// TIA Portal project "Practica_7_p2" (V14)

(* hardware
DEVICE "S7-1200 station_1"  S7-1200 Station
   slot 0: "Rack_0"  S7-1200 Rack  Rack  V1.0
   slot 1: "PLC_1"  CPU 1214C DC/DC/DC  6ES7 214-1AG40-0XB0  V4.2
*)

// ===== PLC "PLC_1"  CPU 1214C DC/DC/DC =====

VAR_GLOBAL   // PLC tag table "Default tag table"
   "G" AT %M0.0 : Bool;
   "R" AT %M0.1 : Bool;
   "LUZ_ROJA" AT %Q0.0 : Bool;
   "LUZ_VERDE" AT %Q0.1 : Bool;
   "OFF" AT %M0.2 : Bool;
   "PM" AT %I0.0 : Bool;
   "PP" AT %I0.1 : Bool;
   "EN" AT %M0.4 : Bool;
END_VAR

DATA_BLOCK "DB_TIMERS_CONFIG"   // DB1
{ S7_Optimized_Access := 'TRUE' }
VERSION : 0.1
   VAR
      TR : Time := T#6s;
      TV : Time := T#5s;
   END_VAR
BEGIN
END_DATA_BLOCK

// folder: System blocks/Program resources

DATA_BLOCK "t_r2v"   // DB2
{ S7_Optimized_Access := 'TRUE' }
AUTHOR : Simatic
FAMILY : IEC
NAME : IEC_TMR
VERSION : 1.0
// stored: InstanceOfName IEC_TIMER
"IEC_TIMER"
BEGIN
END_DATA_BLOCK

DATA_BLOCK "t_v2r"   // DB3
{ S7_Optimized_Access := 'TRUE' }
AUTHOR : Simatic
FAMILY : IEC
NAME : IEC_TMR
VERSION : 1.0
// stored: InstanceOfName IEC_TIMER
"IEC_TIMER"
BEGIN
END_DATA_BLOCK

// folder: (top level)

FUNCTION "FC_SEMAFORO_V1" : Void   // FC1, LAD
{ S7_Optimized_Access := 'TRUE' }
VERSION : 0.1
   VAR_INPUT
      ENABLE : Bool;
      TV : Time;
      TR : Time;
   END_VAR
   VAR_OUTPUT
      LR : Bool;
      LV : Bool;
   END_VAR
   VAR_TEMP   // added for the SCL form of the ladder/FBD networks
      _w1 : Bool;
      _w2 : Bool;
   END_VAR
BEGIN

REGION Network 1
   // INICIALIZACIÓN DE ESTADOS
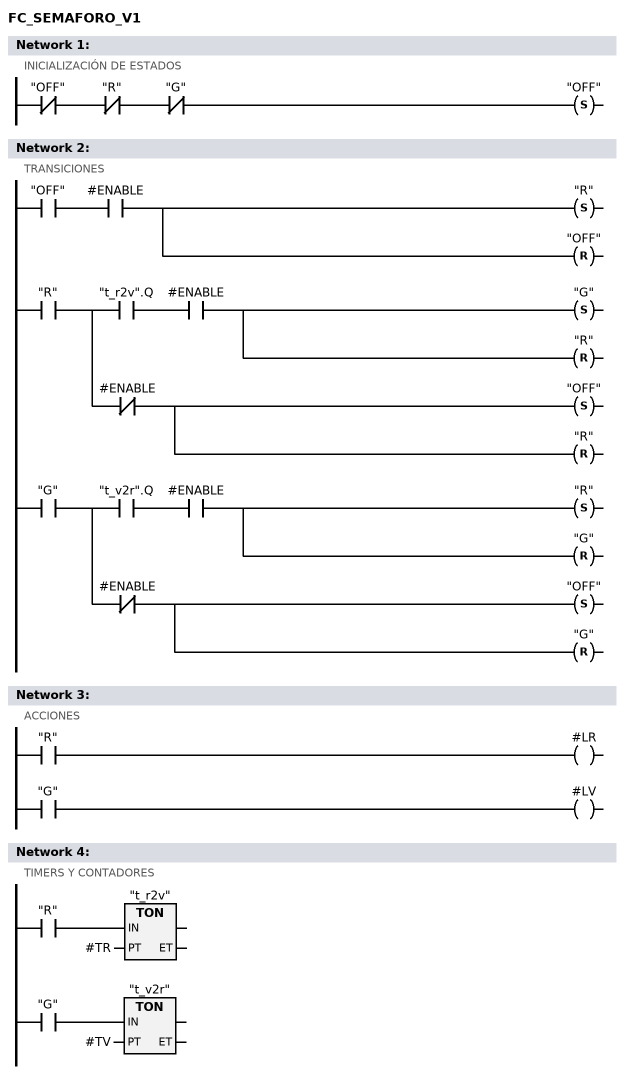
   RUNG wire#powerrail
      I_Contact( "OFF" )
      I_Contact( "R" )
      I_Contact( "G" )
      S_Coil( "OFF" )
   END_RUNG
   // the same network as SCL:
   IF NOT "OFF" AND NOT "R" AND NOT "G" THEN "OFF" := TRUE; END_IF;
END_REGION

REGION Network 2
   // TRANSICIONES
   RUNG wire#powerrail
      Contact( "OFF" )
      Contact( #ENABLE )
      wire#w1
      S_Coil( "R" )
   END_RUNG
   RUNG wire#w1
      R_Coil( "OFF" )
   END_RUNG
   RUNG wire#powerrail
      Contact( "R" )
      wire#w2
      Contact( "t_r2v".Q )
      Contact( #ENABLE )
      wire#w3
      S_Coil( "G" )
   END_RUNG
   RUNG wire#w3
      R_Coil( "R" )
   END_RUNG
   RUNG wire#w2
      I_Contact( #ENABLE )
      wire#w4
      S_Coil( "OFF" )
   END_RUNG
   RUNG wire#w4
      R_Coil( "R" )
   END_RUNG
   RUNG wire#powerrail
      Contact( "G" )
      wire#w5
      Contact( "t_v2r".Q )
      Contact( #ENABLE )
      wire#w6
      S_Coil( "R" )
   END_RUNG
   RUNG wire#w6
      R_Coil( "G" )
   END_RUNG
   RUNG wire#w5
      I_Contact( #ENABLE )
      wire#w7
      S_Coil( "OFF" )
   END_RUNG
   RUNG wire#w7
      R_Coil( "G" )
   END_RUNG
   // the same network as SCL:
   IF "OFF" AND #ENABLE THEN
       "R" := TRUE;
       "OFF" := FALSE;
   END_IF;
   IF "R" AND "t_r2v".Q AND #ENABLE THEN "G" := TRUE; END_IF;
   #_w1 := "R";
   IF "R" AND "t_r2v".Q AND #ENABLE THEN "R" := FALSE; END_IF;
   IF #_w1 AND NOT #ENABLE THEN
       "OFF" := TRUE;
       "R" := FALSE;
   END_IF;
   IF "G" AND "t_v2r".Q AND #ENABLE THEN "R" := TRUE; END_IF;
   #_w2 := "G";
   IF "G" AND "t_v2r".Q AND #ENABLE THEN "G" := FALSE; END_IF;
   IF #_w2 AND NOT #ENABLE THEN
       "OFF" := TRUE;
       "G" := FALSE;
   END_IF;
END_REGION

REGION Network 3
   // ACCIONES
   RUNG wire#powerrail
      Contact( "R" )
      Coil( #LR )
   END_RUNG
   RUNG wire#powerrail
      Contact( "G" )
      Coil( #LV )
   END_RUNG
   // the same network as SCL:
   #LR := "R";
   #LV := "G";
END_REGION

REGION Network 4
   // TIMERS Y CONTADORES
   "t_r2v".TON(IN := "R", PT := #TR);
   "t_v2r".TON(IN := "G", PT := #TV);
END_REGION
END_FUNCTION

ORGANIZATION_BLOCK "Main"   // OB1, LAD, ProgramCycle
TITLE = "Main Program Sweep (Cycle)"
{ S7_Optimized_Access := 'TRUE' }
VERSION : 0.1
   VAR_INPUT
      Initial_Call : Bool;   // Initial call of this OB
      Remanence : Bool;   // =True, if remanent data are available
   END_VAR
BEGIN

REGION Network 1
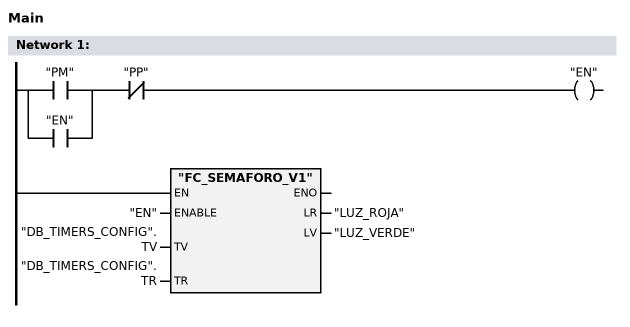
   RUNG wire#powerrail
      Contact( "PM" )
      wire#w1
      I_Contact( "PP" )
      Coil( "EN" )
   END_RUNG
   RUNG wire#powerrail
      Contact( "EN" )
   END_RUNG wire#w1
   RUNG wire#powerrail
      "FC_SEMAFORO_V1"(ENABLE := "EN", TV := "DB_TIMERS_CONFIG".TV, TR := "DB_TIMERS_CONFIG".TR, LR => "LUZ_ROJA", LV => "LUZ_VERDE")
   END_RUNG
   // the same network as SCL:
   "EN" := ("PM" OR "EN") AND NOT "PP";
   "FC_SEMAFORO_V1"(ENABLE := "EN",
                    TV := "DB_TIMERS_CONFIG".TV,
                    TR := "DB_TIMERS_CONFIG".TR,
                    LR => "LUZ_ROJA",
                    LV => "LUZ_VERDE");
END_REGION
END_ORGANIZATION_BLOCK